// SIMATIC S7-200 SMART project (STEP 7-Micro/WIN SMART), CPU ST60

SYMBOL_TABLE V区符号
参数传输成功           V0.0
参数是否更新           V0.1
挡板自动控制完成标志       V0.2
挡板电机开关           V0.3
挡板手动向内           V0.4
挡板手动向外           V0.5
置工件就绪            V0.6
下料电机开关           V0.7
下料前进点动           V1.0
下料后退点动           V1.1
冷却电机开关           V1.2
冷却电机向内           V1.3
冷却电机向外           V1.4
挡板电机查找原点按钮       V11.1
下料电机查找原点按钮       V11.2
冷却电机查找原点按钮       V11.3
挡板自动控制           V11.4
下料下移一个工位         V11.5
下料启动按钮           V11.6
下料手动完成标志         V11.7
回到底部             V12.0
挡板电机子例程          V20.1
挡板电机错误参数         VB21
挡板电机当前位置         VD24
挡板电机当前速度         VD28
挡板电机当前运动方向       V20.2
挡板电机移动位置         VD44
挡板电机速度           VD48
挡板电机移动模式         VB41
挡板电机停止运动轴        V40.1
挡板电机运动方向         V40.2
冷却电机子例程          V60.1
冷却电机错误参数         VB61
冷却电机当前位置         VD64
冷却电机当前速度         VD68
冷却电机当前运动方向       V60.2
冷却电机移动位置         VD84
冷却电机速度           VD88
冷却电机移动模式         VB81
冷却电机停止运动轴        V80.1
冷却电机运动方向         V80.2
下料电机子例程          V100.1
下料电机错误参数         VB101
下料电机当前位置         VD104
下料电机当前速度         VD108
下料电机当前运动方向       V100.2
下料电机移动位置         VD124
下料电机速度           VD128
下料电机移动模式         VB121
下料电机停止运动轴        V120.1
下料电机运动方向         V120.2
上一杆件数据           VD140
当前杆件数据           VD144
下料电机一号工位         VD150
下料电机杆件间距         VD154
下料电机二号工位         VD158
下料电机三号工位         VD162
下料电机四号工位         VD166
下料电机五号工位         VD170
下料电机取小车处         VD174
END_SYMBOL_TABLE

SYMBOL_TABLE 系统符号
Always_On        SM0.0    // 始终接通
END_SYMBOL_TABLE

SYMBOL_TABLE M区符号
挡板超限报警           M0.0
更新配对表            M0.1
挡板步进到位状态位        M0.2
电机是否就绪状态位        M0.3
上料步进到位状态位        M0.4
上料工件有无状态位        M0.5
下料步进到位状态位        M0.6
下料小车到位状态位        M0.7
步进报警信息           M1.0
上料传动故障报警         M1.1
END_SYMBOL_TABLE

ORGANIZATION_BLOCK MAIN:OB1
TITLE=程序注释
BEGIN
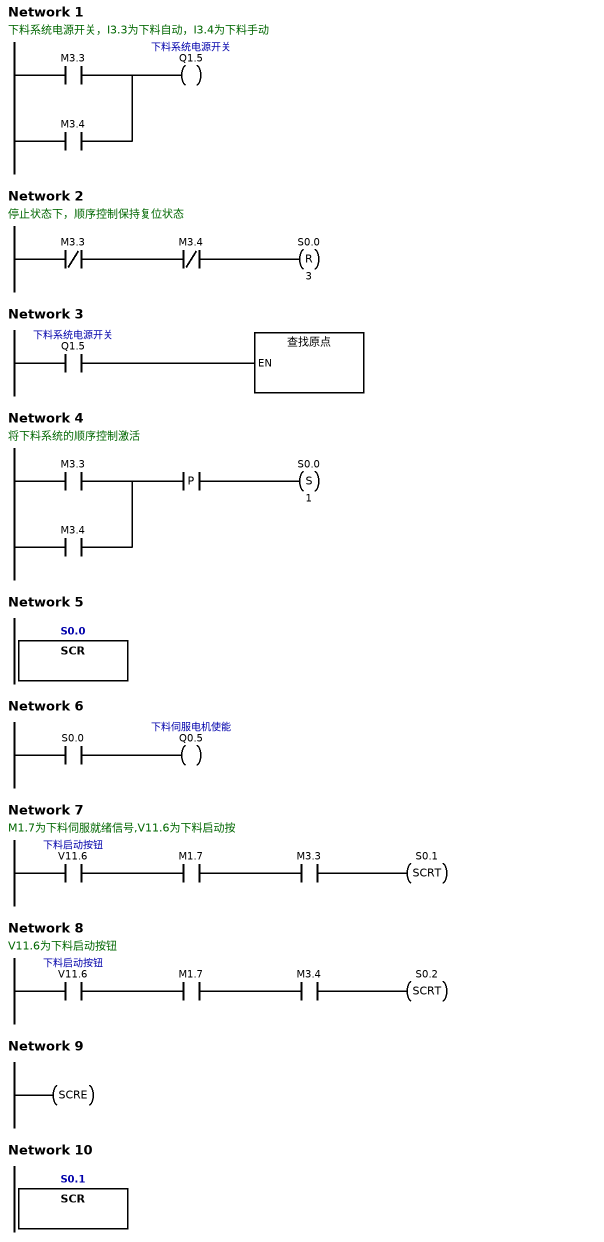
Network 1
// 下料系统电源开关，I3.3为下料自动，I3.4为下料手动
LD     M3.3
O      M3.4
=      下料系统电源开关:Q1.5
Network 2
// 停止状态下，顺序控制保持复位状态
LDN    M3.3
AN     M3.4
R      S0.0, 3
Network 3
LD     下料系统电源开关:Q1.5
CALL   查找原点:SBR5
Network 4
// 将下料系统的顺序控制激活
LD     M3.3
O      M3.4
EU
S      S0.0, 1
Network 5
LSCR   S0.0
Network 6
LD     S0.0
=      下料伺服电机使能:Q0.5
Network 7
// M1.7为下料伺服就绪信号,V11.6为下料启动按
LD     下料启动按钮:V11.6
A      M1.7
A      M3.3
SCRT   S0.1
Network 8
// V11.6为下料启动按钮
LD     下料启动按钮:V11.6
A      M1.7
A      M3.4
SCRT   S0.2
Network 9
SCRE
Network 10
LSCR   S0.1
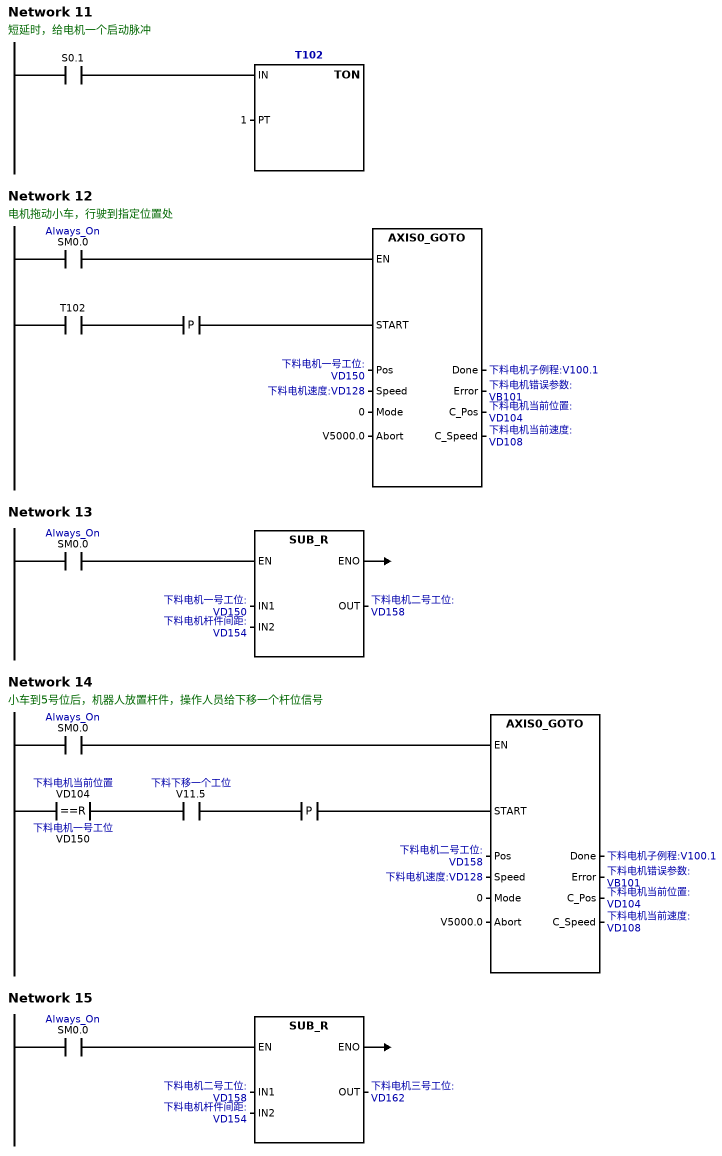
Network 11
// 短延时，给电机一个启动脉冲
LD     S0.1
TON    T102, 1
Network 12
// 电机拖动小车，行驶到指定位置处
LD     Always_On:SM0.0
=      L60.0
LD     T102
EU
=      L63.7
LD     L60.0
CALL   AXIS0_GOTO:SBR3, L63.7, 下料电机一号工位:VD150, 下料电机速度:VD128, 0, V5000.0, 下料电机子例程:V100.1, 下料电机错误参数:VB101, 下料电机当前位置:VD104, 下料电机当前速度:VD108
Network 13
LD     Always_On:SM0.0
MOVR   下料电机一号工位:VD150, 下料电机二号工位:VD158
-R     下料电机杆件间距:VD154, 下料电机二号工位:VD158
Network 14
// 小车到5号位后，机器人放置杆件，操作人员给下移一个杆位信号
LD     Always_On:SM0.0
=      L60.0
LDR=   下料电机当前位置:VD104, 下料电机一号工位:VD150
A      下料下移一个工位:V11.5
EU
=      L63.7
LD     L60.0
CALL   AXIS0_GOTO:SBR3, L63.7, 下料电机二号工位:VD158, 下料电机速度:VD128, 0, V5000.0, 下料电机子例程:V100.1, 下料电机错误参数:VB101, 下料电机当前位置:VD104, 下料电机当前速度:VD108
Network 15
LD     Always_On:SM0.0
MOVR   下料电机二号工位:VD158, 下料电机三号工位:VD162
-R     下料电机杆件间距:VD154, 下料电机三号工位:VD162
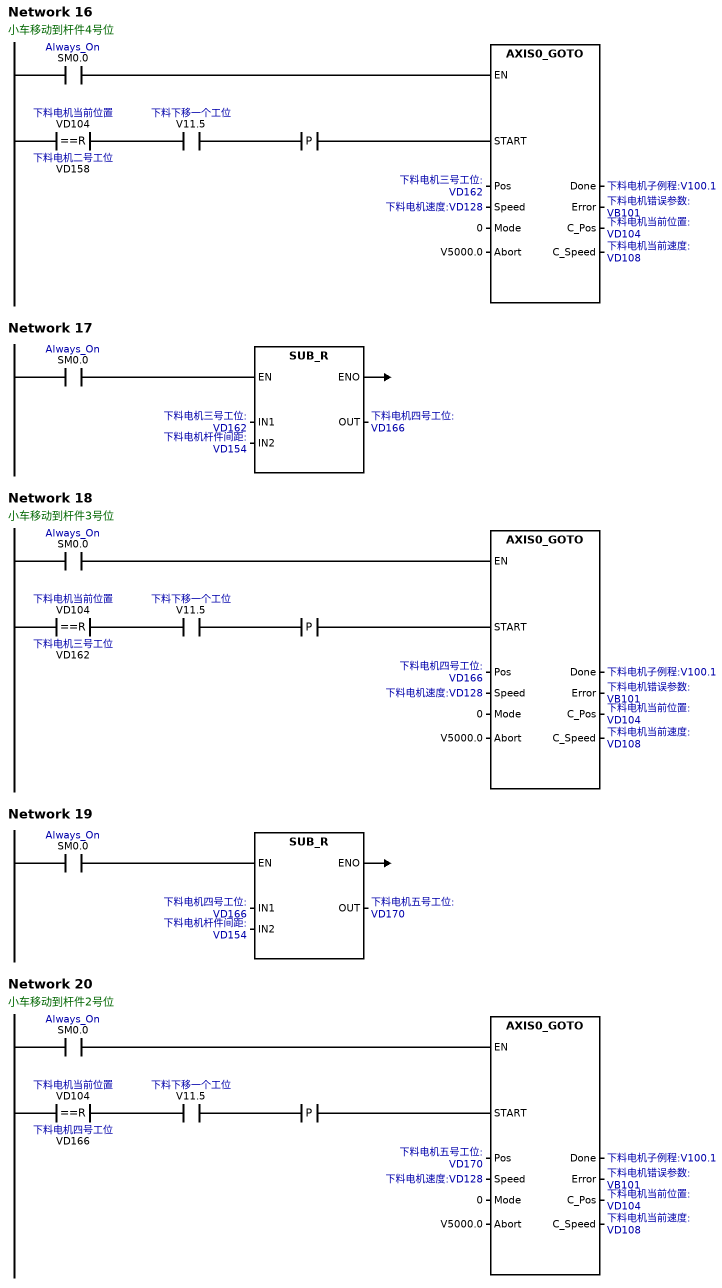
Network 16
// 小车移动到杆件4号位
LD     Always_On:SM0.0
=      L60.0
LDR=   下料电机当前位置:VD104, 下料电机二号工位:VD158
A      下料下移一个工位:V11.5
EU
=      L63.7
LD     L60.0
CALL   AXIS0_GOTO:SBR3, L63.7, 下料电机三号工位:VD162, 下料电机速度:VD128, 0, V5000.0, 下料电机子例程:V100.1, 下料电机错误参数:VB101, 下料电机当前位置:VD104, 下料电机当前速度:VD108
Network 17
LD     Always_On:SM0.0
MOVR   下料电机三号工位:VD162, 下料电机四号工位:VD166
-R     下料电机杆件间距:VD154, 下料电机四号工位:VD166
Network 18
// 小车移动到杆件3号位
LD     Always_On:SM0.0
=      L60.0
LDR=   下料电机当前位置:VD104, 下料电机三号工位:VD162
A      下料下移一个工位:V11.5
EU
=      L63.7
LD     L60.0
CALL   AXIS0_GOTO:SBR3, L63.7, 下料电机四号工位:VD166, 下料电机速度:VD128, 0, V5000.0, 下料电机子例程:V100.1, 下料电机错误参数:VB101, 下料电机当前位置:VD104, 下料电机当前速度:VD108
Network 19
LD     Always_On:SM0.0
MOVR   下料电机四号工位:VD166, 下料电机五号工位:VD170
-R     下料电机杆件间距:VD154, 下料电机五号工位:VD170
Network 20
// 小车移动到杆件2号位
LD     Always_On:SM0.0
=      L60.0
LDR=   下料电机当前位置:VD104, 下料电机四号工位:VD166
A      下料下移一个工位:V11.5
EU
=      L63.7
LD     L60.0
CALL   AXIS0_GOTO:SBR3, L63.7, 下料电机五号工位:VD170, 下料电机速度:VD128, 0, V5000.0, 下料电机子例程:V100.1, 下料电机错误参数:VB101, 下料电机当前位置:VD104, 下料电机当前速度:VD108
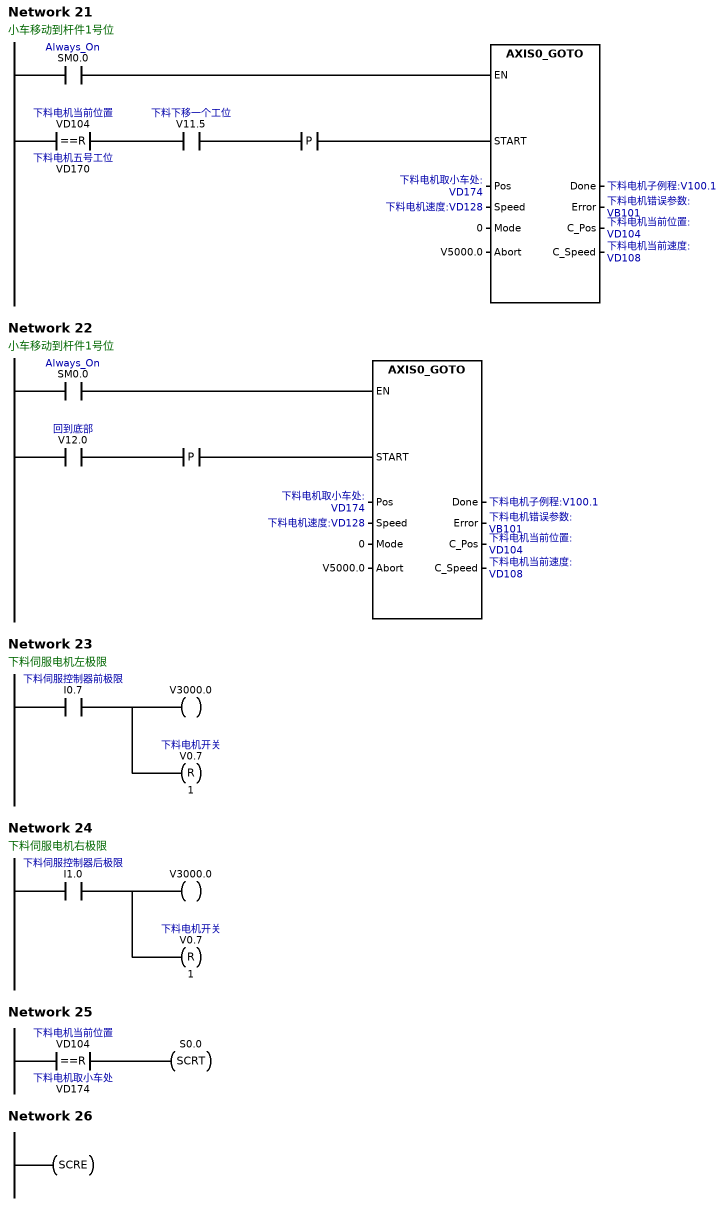
Network 21
// 小车移动到杆件1号位
LD     Always_On:SM0.0
=      L60.0
LDR=   下料电机当前位置:VD104, 下料电机五号工位:VD170
A      下料下移一个工位:V11.5
EU
=      L63.7
LD     L60.0
CALL   AXIS0_GOTO:SBR3, L63.7, 下料电机取小车处:VD174, 下料电机速度:VD128, 0, V5000.0, 下料电机子例程:V100.1, 下料电机错误参数:VB101, 下料电机当前位置:VD104, 下料电机当前速度:VD108
Network 22
// 小车移动到杆件1号位
LD     Always_On:SM0.0
=      L60.0
LD     回到底部:V12.0
EU
=      L63.7
LD     L60.0
CALL   AXIS0_GOTO:SBR3, L63.7, 下料电机取小车处:VD174, 下料电机速度:VD128, 0, V5000.0, 下料电机子例程:V100.1, 下料电机错误参数:VB101, 下料电机当前位置:VD104, 下料电机当前速度:VD108
Network 23
// 下料伺服电机左极限
LD     下料伺服控制器前极限:I0.7
=      V3000.0
R      下料电机开关:V0.7, 1
Network 24
// 下料伺服电机右极限
LD     下料伺服控制器后极限:I1.0
=      V3000.0
R      下料电机开关:V0.7, 1
Network 25
LDR=   下料电机当前位置:VD104, 下料电机取小车处:VD174
SCRT   S0.0
Network 26
SCRE
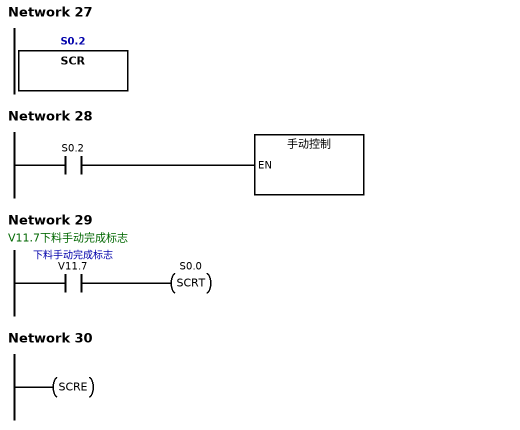
Network 27
LSCR   S0.2
Network 28
LD     S0.2
CALL   手动控制:SBR0
Network 29
// V11.7下料手动完成标志
LD     下料手动完成标志:V11.7
SCRT   S0.0
Network 30
SCRE
END_ORGANIZATION_BLOCK

SUBROUTINE_BLOCK 手动控制:SBR0
TITLE=子程序注释
BEGIN
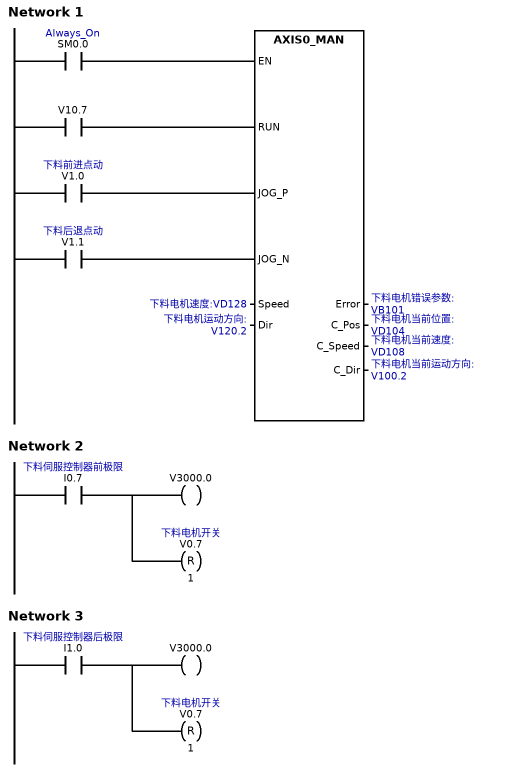
Network 1
LD     Always_On:SM0.0
=      L60.0
LD     V10.7
=      L63.7
LD     下料前进点动:V1.0
=      L63.6
LD     下料后退点动:V1.1
=      L63.5
LD     L60.0
CALL   AXIS0_MAN:SBR2, L63.7, L63.6, L63.5, 下料电机速度:VD128, 下料电机运动方向:V120.2, 下料电机错误参数:VB101, 下料电机当前位置:VD104, 下料电机当前速度:VD108, 下料电机当前运动方向:V100.2
Network 2
LD     下料伺服控制器前极限:I0.7
=      V3000.0
R      下料电机开关:V0.7, 1
Network 3
LD     下料伺服控制器后极限:I1.0
=      V3000.0
R      下料电机开关:V0.7, 1
END_SUBROUTINE_BLOCK

// SBR1: protected block, not included

// SBR2: protected block, not included

// SBR3: protected block, not included

// SBR4: protected block, not included

SUBROUTINE_BLOCK 查找原点:SBR5
TITLE=子程序注释
BEGIN
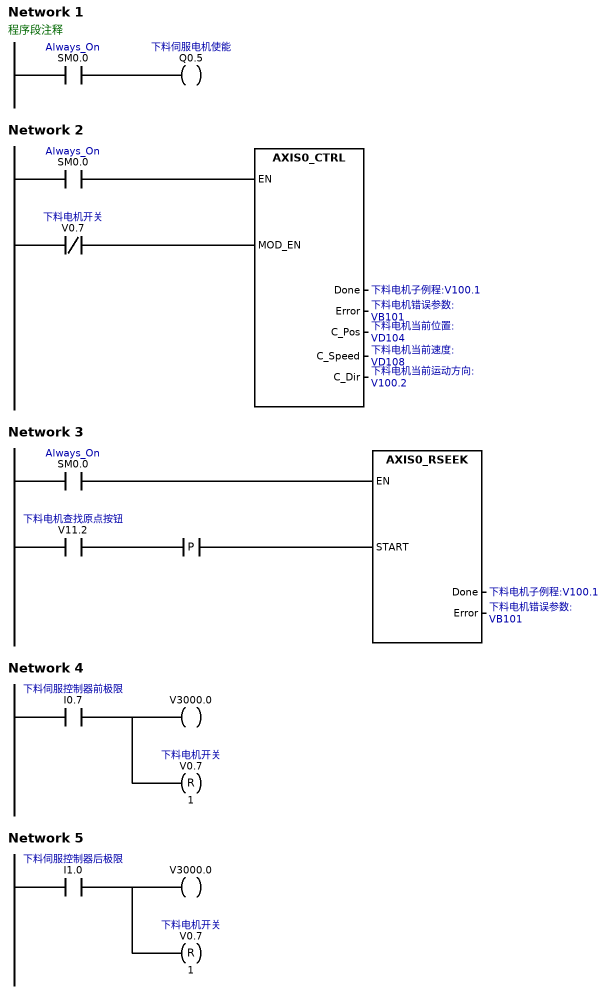
Network 1
// 程序段注释
LD     Always_On:SM0.0
=      下料伺服电机使能:Q0.5
Network 2
LD     Always_On:SM0.0
=      L60.0
LDN    下料电机开关:V0.7
=      L63.7
LD     L60.0
CALL   AXIS0_CTRL:SBR1, L63.7, 下料电机子例程:V100.1, 下料电机错误参数:VB101, 下料电机当前位置:VD104, 下料电机当前速度:VD108, 下料电机当前运动方向:V100.2
Network 3
LD     Always_On:SM0.0
=      L60.0
LD     下料电机查找原点按钮:V11.2
EU
=      L63.7
LD     L60.0
CALL   AXIS0_RSEEK:SBR4, L63.7, 下料电机子例程:V100.1, 下料电机错误参数:VB101
Network 4
LD     下料伺服控制器前极限:I0.7
=      V3000.0
R      下料电机开关:V0.7, 1
Network 5
LD     下料伺服控制器后极限:I1.0
=      V3000.0
R      下料电机开关:V0.7, 1
END_SUBROUTINE_BLOCK
